PROGRAM MAIN
VAR
END_VAR

END_PROGRAM

(* stored: Version 1.1.0.1
   POU MAIN: Id {6966337f-e940-444b-8f58-b318ce9abb69} *)
